// TwinCAT 3 PLC project Lamppu2
// ProgramVersion: 3.1.4026.10
// CompilerDefines: VISU_USEPROPERTYINFO
// libraries:
//   Tc2_Standard, * (Beckhoff Automation GmbH)
//   Tc2_System, * (Beckhoff Automation GmbH)
//   VisuDialogs, * (System)
// project tree:
//   / GlobalTextList.TcGTLO, PlcTask.TcTTO, Visualization Manager.TcVMO (not stored)
//   POUs/ MAIN.TcPOU
//   VISUs/ Visualization.TcVIS
// real-time tasks:
//   TASK PlcTask: cycle T#10ms, priority 20, ADS port 350

CONFIGURATION Lamppu2
    RESOURCE PLC ON TwinCAT3
        TASK PlcTask(INTERVAL := T#10ms, PRIORITY := 20);
        PROGRAM MAIN WITH PlcTask : MAIN;
    END_RESOURCE
END_CONFIGURATION

// ---- POUs/MAIN.TcPOU
PROGRAM MAIN
VAR
	_Lamp		:BOOL;
	_Button1	:BOOL;
	_Button2	:BOOL;
END_VAR

//This program simulates the operation of a lamp, which can be turned on
//by pressing two separate buttons. Both buttons are toggle buttons, so one
//can be pressed after the other. Both buttons have to be pressed to turn
//the light on.

IF _Button1 AND _Button2 THEN
	_Lamp := TRUE;
	
ELSE
	_Lamp := FALSE;
END_IF

END_PROGRAM

// ---- GlobalTextList.TcGTLO
TEXTLIST GlobalTextList
  687 = 'Button 1'
  347 = 'Button 2'
END_TEXTLIST

// ---- VISUs/Visualization.TcVIS
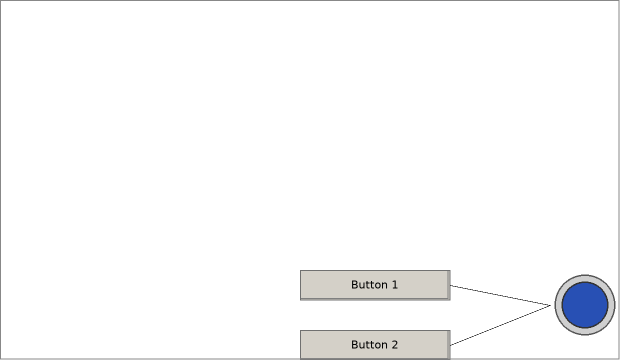
VISUALIZATION Visualization  // 620x360
    Button (300,270 150x30), "Button 1"
        OnMouseClick: toggle MAIN._Button1
    Button (300,330 150x30), "Button 2"
        OnMouseClick: toggle MAIN._Button2
    Lamp1 (550,270 70x70), variable: MAIN._Lamp, style: Lamp-Lamp1-Blue
    Line (450,285) (550,305)
    Line (450,345) (550,305)
END_VISUALIZATION
